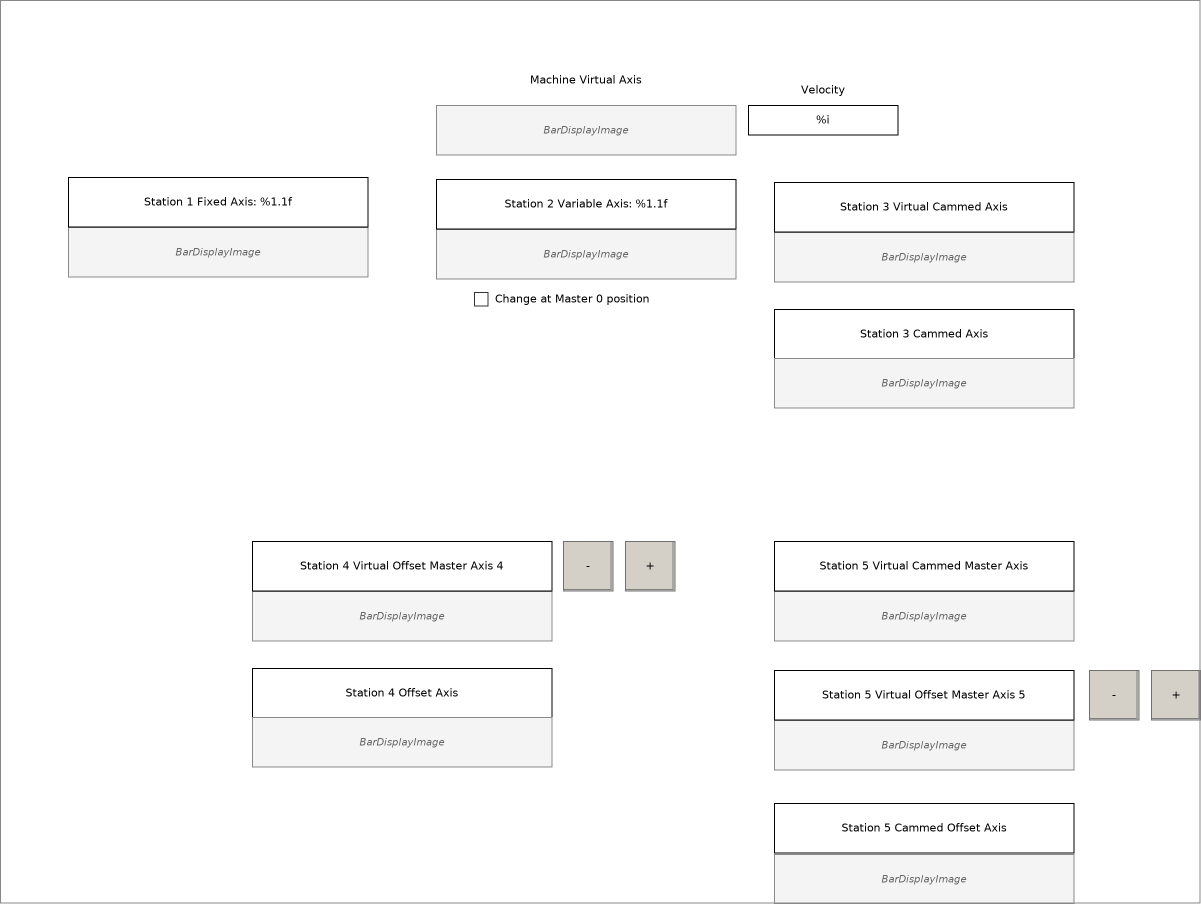
VISUALIZATION V_Operation  // 1201x904
    BarDisplayImage (436,105 300x50), value: MAIN.Machine.MainDrive.MachineVirtualAxis.AxisBase_HMI.Status.ActualPosition, style: BarDisplayImage-Gray, scale format: %.1f, scale 0..1000
    Label (436,55 300x50), "Machine Virtual Axis"
    BarDisplayImage (68,227 300x50), value: MAIN.Machine.Station1.FixedAxis.AxisBase_HMI.Status.ActualPosition, style: BarDisplayImage-Gray, scale format: %.1f, scale 0..1000
    Rectangle (68,177 300x50), "Station 1 Fixed Axis: %1.1f", text variable: MAIN.Machine.Station1.FixedAxis.BasicSlaveAxis._RatioMaster1
    BarDisplayImage (436,229 300x50), value: MAIN.Machine.Station2.VariableAxis.AxisBase_HMI.Status.ActualPosition, style: BarDisplayImage-Gray, scale format: %.1f, scale -2000..2000
    Rectangle (436,179 300x50), "Station 2 Variable Axis: %1.1f", text variable: MAIN.Machine.Station2.variableGearRatio
        OnMouseClick: write the text variable via VisuDialogs.Numpad, min -2.0, max 2.0
    BarDisplayImage (774,232 300x50), value: MAIN.Machine.Station3.VirtualCammedAxis.AxisBase_HMI.Status.ActualPosition, style: BarDisplayImage-Gray, scale format: %.1f, scale 0..100
    Rectangle (774,182 300x50), "Station 3 Virtual Cammed Axis", text variable: MAIN.Machine.Station2.VariableAxis.BasicSlaveAxis._RatioMaster1
    Rectangle (774,309 300x50), "Station 3 Cammed Axis", text variable: MAIN.Machine.Station3.CammedAxis.AxisBase_HMI.Status.ActualPosition
    BarDisplayImage (774,358 300x50), value: MAIN.Machine.Station3.CammedAxis.AxisBase_HMI.Status.ActualPosition, style: BarDisplayImage-Gray, scale format: %.1f, scale 0..150
    BarDisplayImage (252,591 300x50), value: MAIN.Machine.Station4.VirtualOffsetMasterAxis.AxisBase_HMI.Status.ActualPosition, style: BarDisplayImage-Gray, scale format: %.1f, scale 0..1000
    Rectangle (252,541 300x50), "Station 4 Virtual Offset Master Axis 4", text variable: MAIN.Machine.Station2.VariableAxis.BasicSlaveAxis._RatioMaster1
    Rectangle (252,668 300x50), "Station 4 Offset Axis", text variable: MAIN.Machine.Station3.CammedAxis.AxisBase_HMI.Status.ActualPosition
    BarDisplayImage (252,717 300x50), value: MAIN.Machine.Station4.OffsetAxis.AxisBase_HMI.Status.ActualPosition, style: BarDisplayImage-Gray, scale format: %.1f, scale 0..2000
    BarDisplayImage (774,591 300x50), value: MAIN.Machine.Station5.VirtualCammedMasterAxis.AxisBase_HMI.Status.ActualPosition, style: BarDisplayImage-Gray, scale format: %.1f, scale 0..100
    Rectangle (774,541 300x50), "Station 5 Virtual Cammed Master Axis", text variable: MAIN.Machine.Station2.VariableAxis.BasicSlaveAxis._RatioMaster1
    Rectangle (774,803 300x50), "Station 5 Cammed Offset Axis", text variable: MAIN.Machine.Station3.CammedAxis.AxisBase_HMI.Status.ActualPosition
    BarDisplayImage (774,720 300x50), value: MAIN.Machine.Station5.VirtualOffsetMasterAxis.AxisBase_HMI.Status.ActualPosition, style: BarDisplayImage-Gray, scale format: %.1f, scale 0..1000
    Rectangle (774,670 300x50), "Station 5 Virtual Offset Master Axis 5", text variable: MAIN.Machine.Station2.VariableAxis.BasicSlaveAxis._RatioMaster1
    BarDisplayImage (774,854 300x50), value: MAIN.Machine.Station5.CammedOffsetAxis.AxisBase_HMI.Status.ActualPosition, style: BarDisplayImage-Gray, scale format: %.1f, scale 0..1000
    Rectangle (748,105 150x30), "%i", text variable: MAIN.Machine.MainDrive.MachineVirtualAxis.BasicAxis._Velocity
        OnMouseClick: write the text variable via VisuDialogs.Numpad, min 0, max 100
    Checkbox (472,284 229x30), "Change at Master 0 position", variable: MAIN.Machine.Station2.sync
    Label (748,75 150x30), "Velocity"
    Button (563,541 50x50), "-"
        tap MAIN.Machine.Station4.V_OffsetREV
    Button (625,541 50x50), "+"
        tap MAIN.Machine.Station4.V_OffsetFWD
    Button (1089,670 50x50), "-"
        tap MAIN.Machine.Station5.V_OffsetREV
    Button (1151,670 50x50), "+"
        tap MAIN.Machine.Station5.V_OffsetFWD
END_VISUALIZATION

(* stored: Version 1.1.0.1, ProductVersion 3.1.4024.13
   Visu V_Operation: Id {3e2ce8b6-2101-4d59-b9d5-e25ff74cf65e} *)
